TYPE E_CRYO_BIN_CTRL_ACTION :
(
	NONE := 0,
	OFF,
	ON
);
END_TYPE

(* stored: Version 1.1.0.1, ProductVersion 3.1.4024.9
   DUT E_CRYO_BIN_CTRL_ACTION: Id {32f4559b-30e4-47e6-bd29-c794820ef9e9} *)
